// TIA Portal V20 export
DATA_BLOCK "ControlNodes"   // DB49
// stored: MemoryReserve 100, Namespace Unit1.Em5
   VAR
      em : "LAF_typeEmControlNode";
      emstate { S7_SetPoint := 'True'} : "LUC_typeStates";
      cm : "Unit1.Em5.typeCmControlNode";
      citiMap : Struct
         PMC : "LER_PMC_Input_Data";
         FlexNet { S7_SetPoint := 'True'} : "LER_FlexNet_Data";
      END_STRUCT;
      transferPnPLeft : "Unit1.Em5.typeSequenceControlNode_transferPnPLeft";
      transferPnPRight : "Unit1.Em5.typeSequenceControlNode_transferPnPRight";
      GRnR_TransferPnP : "Unit1.Em5.typeSequenceControlNode_GRnR";
      emData : "Unit1.Em5.typeEmDataControlNode";
      SpecialFunctionMode : Struct
         DryRun : Struct
            JRdetectPV : Array[0..15] of Bool;
         END_STRUCT;
      END_STRUCT;
      cmTransferPnPLeftSafetyPin : "LBC_typeDigitalSignalControlNode";
      cmTransferPnPLeftJRDetect : "LBC_typeDigitalSignalControlNode";
      cmTransferPnPRightSafetyPin : "LBC_typeDigitalSignalControlNode";
      cmTransferPnPRightJRDetect : "LBC_typeDigitalSignalControlNode";
      cmTransferPnPLeftAxisX : "LBC_typeAxis64PosControlNode";
      cmTransferPnPLeftAxisY : "LBC_typeAxis64PosControlNode";
      cmTransferPnPLeftAxisZ : "LBC_typeAxis64PosControlNode";
      cmTransferPnPRightAxisX : "LBC_typeAxis64PosControlNode";
      cmTransferPnPRightAxisY : "LBC_typeAxis64PosControlNode";
      cmTransferPnPRightAxisZ : "LBC_typeAxis64PosControlNode";
      cmTransferPnPLeftClampOpenClose : "LBC_typeTwoWayActuatorControlNode";
      cmTransferPnPRightClampOpenClose : "LBC_typeTwoWayActuatorControlNode";
   END_VAR
BEGIN
END_DATA_BLOCK
